(* IEC 61131-3 sources: heating/Heating/src/hw_lib, 2 files *)

(* ---- I2HAA.iecst ---- *)
FUNCTION I2HAA

	VAR_INPUT
		fd : DINT := -1;
		address : INT := 16#0b;
		channel : SINT := 0;
		value : UINT;
	END_VAR

	VAR
		num_bytes : LINT := -1;
		data : ARRAY[0 .. 63] OF BYTE;
		data_len : INT := 3;

		checked_value : UINT := 0;

		I2C_SLAVE : DINT := 1795; /* a constant from the Linux kernel */
	END_VAR;

	IF value > 1023 THEN
		checked_value := 1023;
	ELSE
		checked_value := value;
	END_IF;

	IF fd >= 0 AND value >= 0 AND value < 1024 THEN
		System_ioctl(fd := fd, request := I2C_SLAVE, data := address, ENO => ENO);
		IF ENO THEN
			data[0] := TO_BYTE(channel);
			data[2] := TO_BYTE(checked_value / 256); /* high byte */
			data[1] := TO_BYTE(checked_value - TO_UINT(data[2]) * 256);  /* low byte */
			num_bytes := System_write(fd := fd, count := data_len, data := data, ENO => ENO);
			IF num_bytes <> data_len THEN
				ENO := FALSE;
			END_IF;
		END_IF;
	ELSE
		ENO := FALSE;
	END_IF;

END_FUNCTION

(* ---- I2HAE.iecst ---- *)
FUNCTION I2HAE : ARRAY[0..4] OF UINT /* 5 channels with 10 bits each */

	VAR_INPUT
		fd : DINT := -1;
		address : INT := 16#0b;
	END_VAR

	VAR
		num_bytes : LINT := -1; /* number of bytes read from bus device */
		cnt : INT := 0;
		data : ARRAY[0 .. 63] OF BYTE;

		I2C_SLAVE : DINT := 1795; /* a constant from the Linux kernel */

		num_channels : INT := 5;
		data_len : INT := 11;
	END_VAR

	IF fd >= 0 THEN
		System_ioctl(fd := fd, request := I2C_SLAVE, data := address, ENO => ENO);
		IF ENO THEN
			num_bytes := Posix_read(fd := fd, count := data_len /* 11 bytes at once(!) */, data => data, ENO => ENO);

			IF ENO AND num_bytes = data_len THEN
				FOR cnt := 0 TO num_channels - 1 BY 1 DO
					I2HAE[cnt] := TO_UINT(data[1 + cnt * 2]) + TO_UINT(data[2 + cnt * 2]) * 256;
				END_FOR;
			END_IF;
		END_IF;
	ELSE
		ENO := FALSE;
	END_IF;

END_FUNCTION
